TYPE GearingAxis :
STRUCT
	AXIS 	    : AXIS_REF;
	RATIO 	    : LREAL;
END_STRUCT
END_TYPE

(* stored: Version 1.1.0.1, ProductVersion 3.1.4022.12
   DUT GearingAxis: Id {13c02ac5-dbb3-42fb-94f9-0b789cdb7841} *)
